// TIA Portal V16 export
// export: Created 2023-10-30T22:43:51.0597784Z, ExportSetting WithDefaults, DisplayName Totally Integrated Automation Portal, DisplayVersion V16, DisplayName TIA Portal Version Control Interface, DisplayVersion V16, DisplayName TIA Portal Openness, DisplayVersion V16, DisplayName SINAMICS Startdrive Advanced, DisplayVersion V16, DisplayName SINAMICS Startdrive G130, G150, S120, S150, SINAMICS MV, S210, DisplayVersion V16, DisplayName SINAMICS Startdrive G110M, G120, G120C, G120D, G120P, DisplayVersion V16, DisplayName STEP 7 Professional, DisplayVersion V16, DisplayName STEP 7 Safety, DisplayVersion V16, DisplayName WinCC Professional, DisplayVersion V16
DATA_BLOCK "Modbus_Comm_Load_DB"   // DB5
// stored: AutoNumber true, DBAccessibleFromOPCUA true, InstanceOfName Modbus_Comm_Load, OfSystemLibElement Modbus_Comm_Load, OfSystemLibVersion 3.1
"Modbus_Comm_Load"
   // VAR_INPUT
   //    REQ : Bool;
   //    PORT : PORT;
   //    BAUD : UDInt;
   //    PARITY : UInt;
   //    FLOW_CTRL : UInt;
   //    RTS_ON_DLY : UInt;
   //    RTS_OFF_DLY : UInt;
   //    RESP_TO : UInt;
   // END_VAR
   // VAR_OUTPUT
   //    DONE : Bool;
   //    ERROR : Bool;
   //    STATUS : Word;
   // END_VAR
   // VAR_IN_OUT
   //    MB_DB : P2P_MB_BASE;
   // END_VAR
   // VAR
   //    ICHAR_GAP : Word;
   //    RETRIES : Word;
   //    MODE : USInt := 16#04;
   //    LINE_PRE : USInt;
   //    BRK_DET : USInt;
   //    EN_DIAG_ALARM : Bool;
   //    STOP_BITS : USInt;
   //    EN_SUPPLY_VOLT : Bool;
   //    b_e_REQ : Bool;
   //    y_state : SInt;
   //    Send_Config { S7_SetPoint := 'True'} : Send_Config;
   //    Receive_Config { S7_SetPoint := 'True'} : Receive_Config;
   //    Receive_Conditions { S7_SetPoint := 'True'} : Receive_Conditions;
   //    WRREC { S7_SetPoint := 'True'} : WRREC;
   //    RDREC { S7_SetPoint := 'True'} : RDREC;
   //    port_w_record { ExternalVisible := 'False'; S7_SetPoint := 'True'} : P2P_MB_PortData;
   //    err_record { ExternalVisible := 'False'; S7_SetPoint := 'True'} : P2P_RdEstat;
   //    ftrs_w_record { ExternalVisible := 'False'; S7_SetPoint := 'True'} : P2P_FeaturesData;
   //    wlen : UInt;
   // END_VAR
BEGIN
END_DATA_BLOCK
